(* Logix 5000 project; controller cal1632 1756-L62 rev 16.20; software revision 16.05; part 38 of 61 *)
(* tags used below, declared in another part *)
   p23r17 : routine;
   FAULT : BOOL;
   HMI : BOOL;
   p01r09_pb_global_reset : BOOL;
   p02_real_from_hmi : hmi_real;
   p23_ai_lfl : REAL;
   p23_ai_metering_roll_amps : REAL;
   p23_ai_metering_roll_hz : REAL;
   p23_ai_metering_roll_speed_fpm : REAL;
   p23_ai_prs : REAL;
   p23_ai_servo_ds_position : REAL;
   p23_ai_servo_ds_torque : REAL;
   p23_ai_servo_os_position : REAL;
   p23_ai_servo_os_torque : REAL;
   p23_ai_servo_os_velocity : REAL;
   p23_ai_supply_amps : REAL;
   p23_ai_supply_hz : REAL;
   p23_ai_supply_rpm : REAL;
   p23_dint_to_hmi : DINT[32];
   p23_param_lfl_hhl : REAL;
   p23_param_lfl_hl : REAL;
   p23_param_zone_pressure : REAL;
   p23_real_to_hmi : REAL[112];
   p23r02 : routine;
   p23r06 : routine;
   p23r06_timer_fault : TIMER[4];
   p23r06_timer_warning : TIMER[4];
   p23r07 : routine;
   p23r07_timer_fault : TIMER[4];
   p23r07_timer_warning : TIMER[4];
   p23r08 : routine;
   p23r08_timer_fault : TIMER[4];
   p23r08_timer_warning : TIMER[4];
   p23r11 : routine;
   p23r12 : routine;
   p23r13 : routine;
   p23r15 : routine;
(* P23_Impreg, continued *)

ROUTINE R06_Real_to_HMI   (* ladder *)
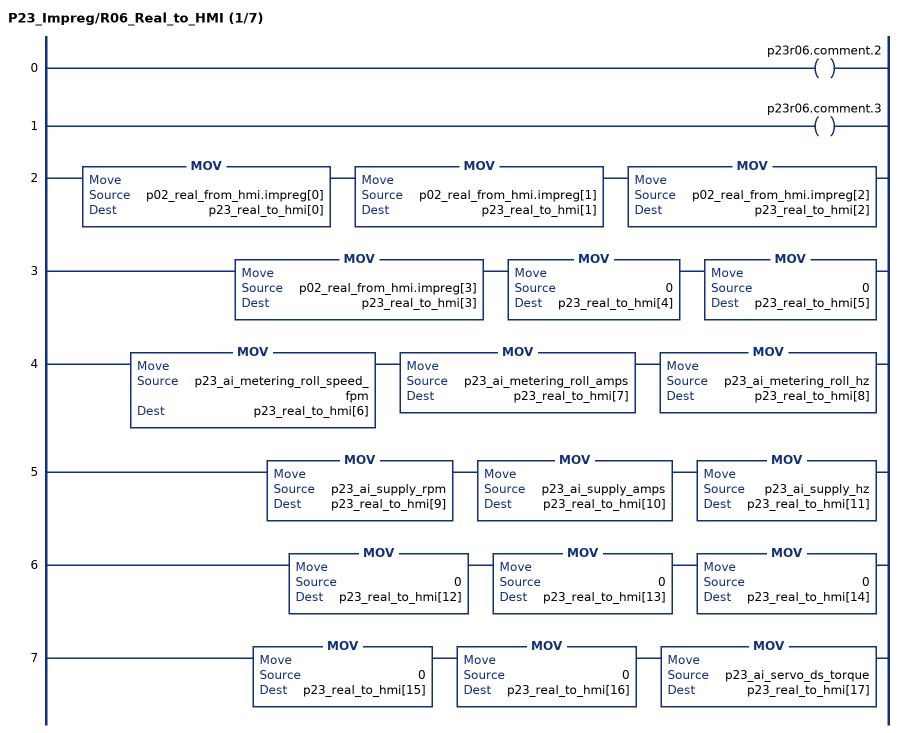
   0: OTE(p23r06.comment.2);
   1: OTE(p23r06.comment.3);
   2: MOV(p02_real_from_hmi.impreg[0],p23_real_to_hmi[0])MOV(p02_real_from_hmi.impreg[1],p23_real_to_hmi[1])MOV(p02_real_from_hmi.impreg[2],p23_real_to_hmi[2]);
   3: MOV(p02_real_from_hmi.impreg[3],p23_real_to_hmi[3])MOV(0,p23_real_to_hmi[4])MOV(0,p23_real_to_hmi[5]);
   4: MOV(p23_ai_metering_roll_speed_fpm,p23_real_to_hmi[6])MOV(p23_ai_metering_roll_amps,p23_real_to_hmi[7])MOV(p23_ai_metering_roll_hz,p23_real_to_hmi[8]);
   5: MOV(p23_ai_supply_rpm,p23_real_to_hmi[9])MOV(p23_ai_supply_amps,p23_real_to_hmi[10])MOV(p23_ai_supply_hz,p23_real_to_hmi[11]);
   6: MOV(0,p23_real_to_hmi[12])MOV(0,p23_real_to_hmi[13])MOV(0,p23_real_to_hmi[14]);
   7: MOV(0,p23_real_to_hmi[15])MOV(0,p23_real_to_hmi[16])MOV(p23_ai_servo_ds_torque,p23_real_to_hmi[17]);
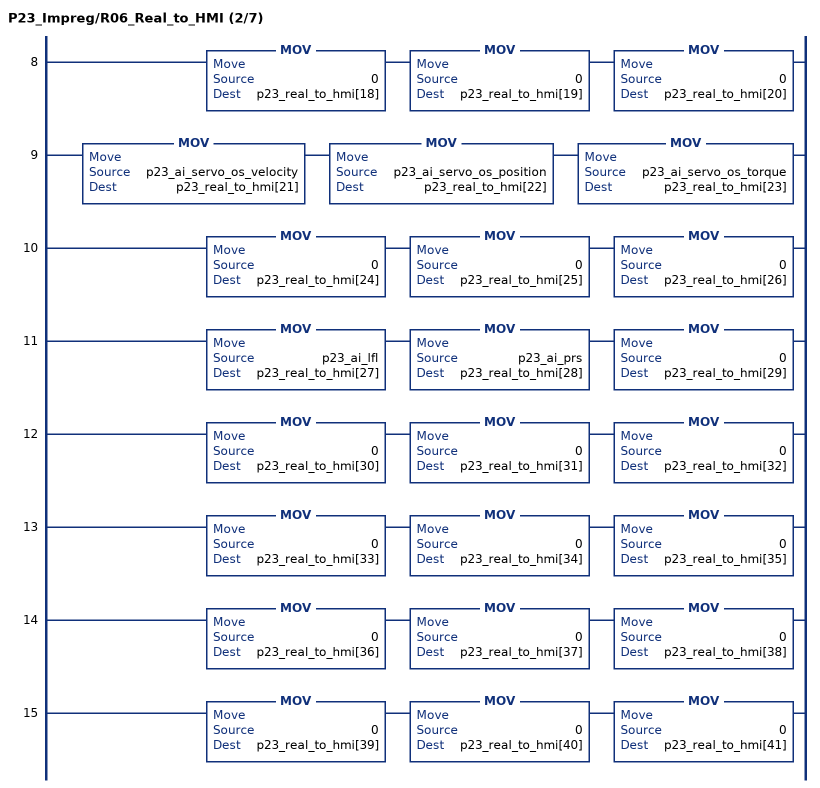
   8: MOV(0,p23_real_to_hmi[18])MOV(0,p23_real_to_hmi[19])MOV(0,p23_real_to_hmi[20]);
   9: MOV(p23_ai_servo_os_velocity,p23_real_to_hmi[21])MOV(p23_ai_servo_os_position,p23_real_to_hmi[22])MOV(p23_ai_servo_os_torque,p23_real_to_hmi[23]);
   10: MOV(0,p23_real_to_hmi[24])MOV(0,p23_real_to_hmi[25])MOV(0,p23_real_to_hmi[26]);
   11: MOV(p23_ai_lfl,p23_real_to_hmi[27])MOV(p23_ai_prs,p23_real_to_hmi[28])MOV(0,p23_real_to_hmi[29]);
   12: MOV(0,p23_real_to_hmi[30])MOV(0,p23_real_to_hmi[31])MOV(0,p23_real_to_hmi[32]);
   13: MOV(0,p23_real_to_hmi[33])MOV(0,p23_real_to_hmi[34])MOV(0,p23_real_to_hmi[35]);
   14: MOV(0,p23_real_to_hmi[36])MOV(0,p23_real_to_hmi[37])MOV(0,p23_real_to_hmi[38]);
   15: MOV(0,p23_real_to_hmi[39])MOV(0,p23_real_to_hmi[40])MOV(0,p23_real_to_hmi[41]);
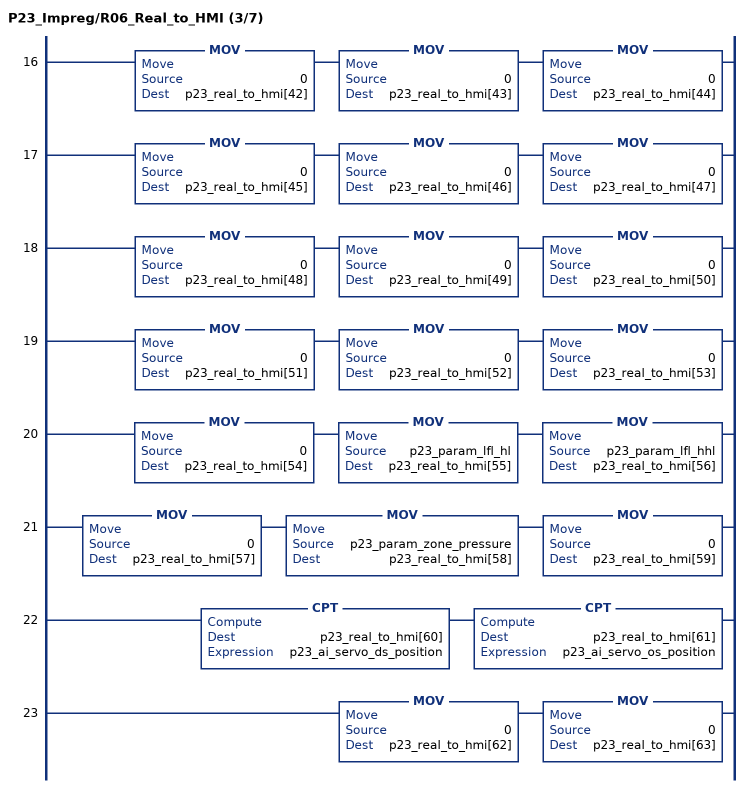
   16: MOV(0,p23_real_to_hmi[42])MOV(0,p23_real_to_hmi[43])MOV(0,p23_real_to_hmi[44]);
   17: MOV(0,p23_real_to_hmi[45])MOV(0,p23_real_to_hmi[46])MOV(0,p23_real_to_hmi[47]);
   18: MOV(0,p23_real_to_hmi[48])MOV(0,p23_real_to_hmi[49])MOV(0,p23_real_to_hmi[50]);
   19: MOV(0,p23_real_to_hmi[51])MOV(0,p23_real_to_hmi[52])MOV(0,p23_real_to_hmi[53]);
   20: MOV(0,p23_real_to_hmi[54])MOV(p23_param_lfl_hl,p23_real_to_hmi[55])MOV(p23_param_lfl_hhl,p23_real_to_hmi[56]);
   21: MOV(0,p23_real_to_hmi[57])MOV(p23_param_zone_pressure,p23_real_to_hmi[58])MOV(0,p23_real_to_hmi[59]);
   22: CPT(p23_real_to_hmi[60],p23_ai_servo_ds_position)CPT(p23_real_to_hmi[61],p23_ai_servo_os_position);
   23: MOV(0,p23_real_to_hmi[62])MOV(0,p23_real_to_hmi[63]);
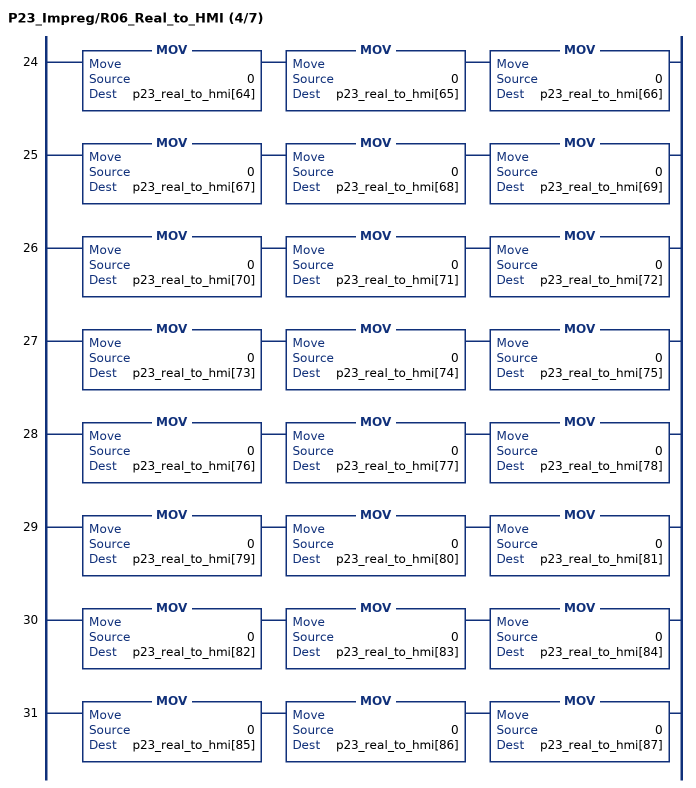
   24: MOV(0,p23_real_to_hmi[64])MOV(0,p23_real_to_hmi[65])MOV(0,p23_real_to_hmi[66]);
   25: MOV(0,p23_real_to_hmi[67])MOV(0,p23_real_to_hmi[68])MOV(0,p23_real_to_hmi[69]);
   26: MOV(0,p23_real_to_hmi[70])MOV(0,p23_real_to_hmi[71])MOV(0,p23_real_to_hmi[72]);
   27: MOV(0,p23_real_to_hmi[73])MOV(0,p23_real_to_hmi[74])MOV(0,p23_real_to_hmi[75]);
   28: MOV(0,p23_real_to_hmi[76])MOV(0,p23_real_to_hmi[77])MOV(0,p23_real_to_hmi[78]);
   29: MOV(0,p23_real_to_hmi[79])MOV(0,p23_real_to_hmi[80])MOV(0,p23_real_to_hmi[81]);
   30: MOV(0,p23_real_to_hmi[82])MOV(0,p23_real_to_hmi[83])MOV(0,p23_real_to_hmi[84]);
   31: MOV(0,p23_real_to_hmi[85])MOV(0,p23_real_to_hmi[86])MOV(0,p23_real_to_hmi[87]);
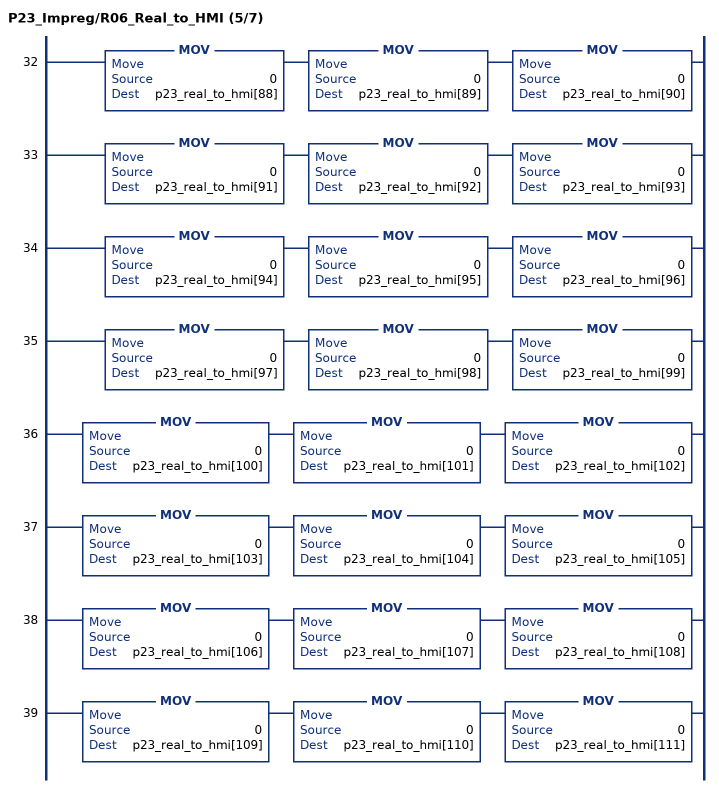
   32: MOV(0,p23_real_to_hmi[88])MOV(0,p23_real_to_hmi[89])MOV(0,p23_real_to_hmi[90]);
   33: MOV(0,p23_real_to_hmi[91])MOV(0,p23_real_to_hmi[92])MOV(0,p23_real_to_hmi[93]);
   34: MOV(0,p23_real_to_hmi[94])MOV(0,p23_real_to_hmi[95])MOV(0,p23_real_to_hmi[96]);
   35: MOV(0,p23_real_to_hmi[97])MOV(0,p23_real_to_hmi[98])MOV(0,p23_real_to_hmi[99]);
   36: MOV(0,p23_real_to_hmi[100])MOV(0,p23_real_to_hmi[101])MOV(0,p23_real_to_hmi[102]);
   37: MOV(0,p23_real_to_hmi[103])MOV(0,p23_real_to_hmi[104])MOV(0,p23_real_to_hmi[105]);
   38: MOV(0,p23_real_to_hmi[106])MOV(0,p23_real_to_hmi[107])MOV(0,p23_real_to_hmi[108]);
   39: MOV(0,p23_real_to_hmi[109])MOV(0,p23_real_to_hmi[110])MOV(0,p23_real_to_hmi[111]);
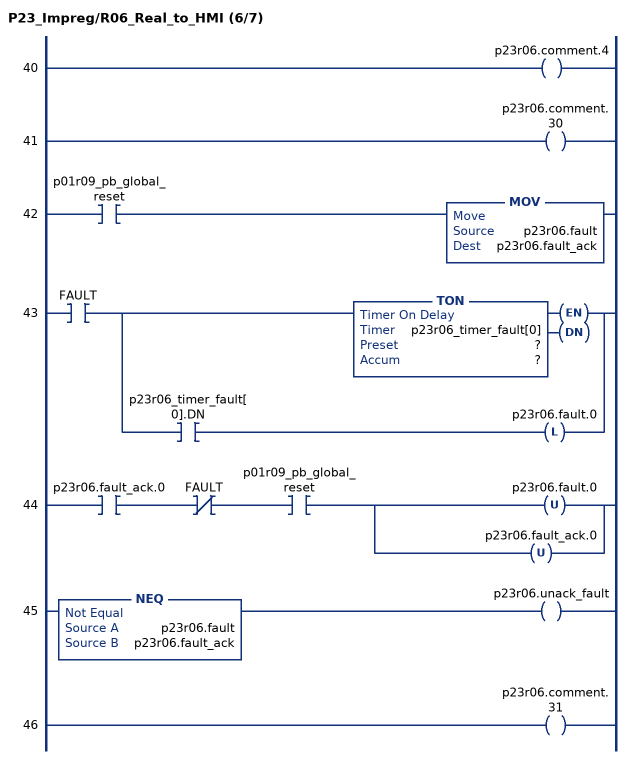
   40: OTE(p23r06.comment.4);
   41: OTE(p23r06.comment.30);
   42: XIC(p01r09_pb_global_reset)MOV(p23r06.fault,p23r06.fault_ack);
   43: XIC(FAULT)[TON(p23r06_timer_fault[0],?,?) ,XIC(p23r06_timer_fault[0].DN) OTL(p23r06.fault.0) ];
   44: XIC(p23r06.fault_ack.0)XIO(FAULT)XIC(p01r09_pb_global_reset)[OTU(p23r06.fault.0) ,OTU(p23r06.fault_ack.0) ];
   45: NEQ(p23r06.fault,p23r06.fault_ack)OTE(p23r06.unack_fault);
   46: OTE(p23r06.comment.31);
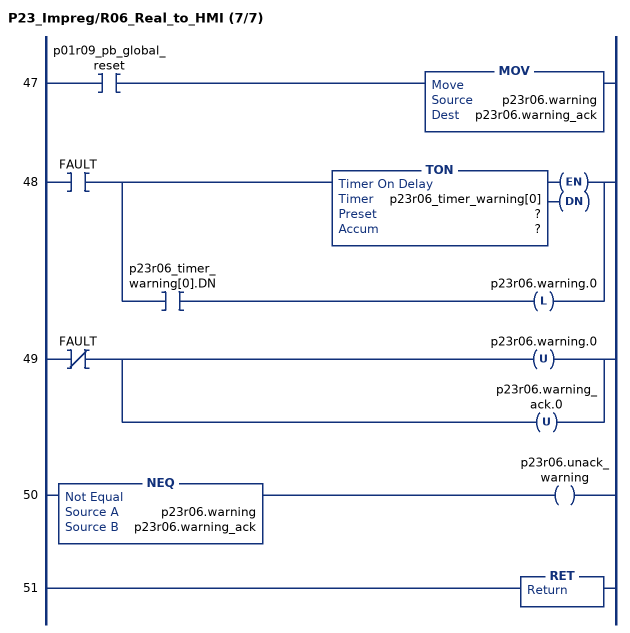
   47: XIC(p01r09_pb_global_reset)MOV(p23r06.warning,p23r06.warning_ack);
   48: XIC(FAULT)[TON(p23r06_timer_warning[0],?,?) ,XIC(p23r06_timer_warning[0].DN) OTL(p23r06.warning.0) ];
   49: XIO(FAULT)[OTU(p23r06.warning.0) ,OTU(p23r06.warning_ack.0) ];
   50: NEQ(p23r06.warning,p23r06.warning_ack)OTE(p23r06.unack_warning);
   51: RET();
END_ROUTINE

ROUTINE R07_Alarms   (* ladder *)
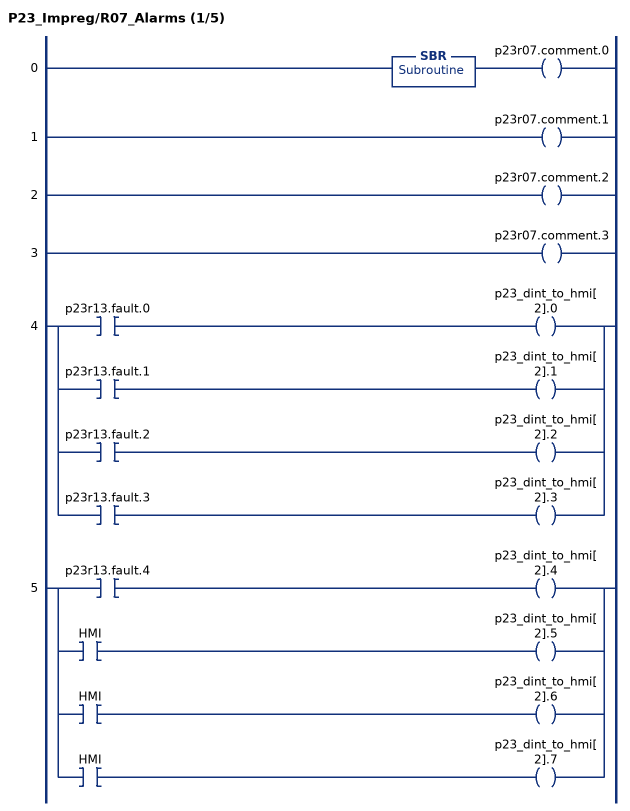
   0: SBR()OTE(p23r07.comment.0);
   1: OTE(p23r07.comment.1);
   2: OTE(p23r07.comment.2);
   3: OTE(p23r07.comment.3);
   4: [XIC(p23r13.fault.0) OTE(p23_dint_to_hmi[2].0) ,XIC(p23r13.fault.1) OTE(p23_dint_to_hmi[2].1) ,XIC(p23r13.fault.2) OTE(p23_dint_to_hmi[2].2) ,XIC(p23r13.fault.3) OTE(p23_dint_to_hmi[2].3) ];
   5: [XIC(p23r13.fault.4) OTE(p23_dint_to_hmi[2].4) ,XIC(HMI) OTE(p23_dint_to_hmi[2].5) ,XIC(HMI) OTE(p23_dint_to_hmi[2].6) ,XIC(HMI) OTE(p23_dint_to_hmi[2].7) ];
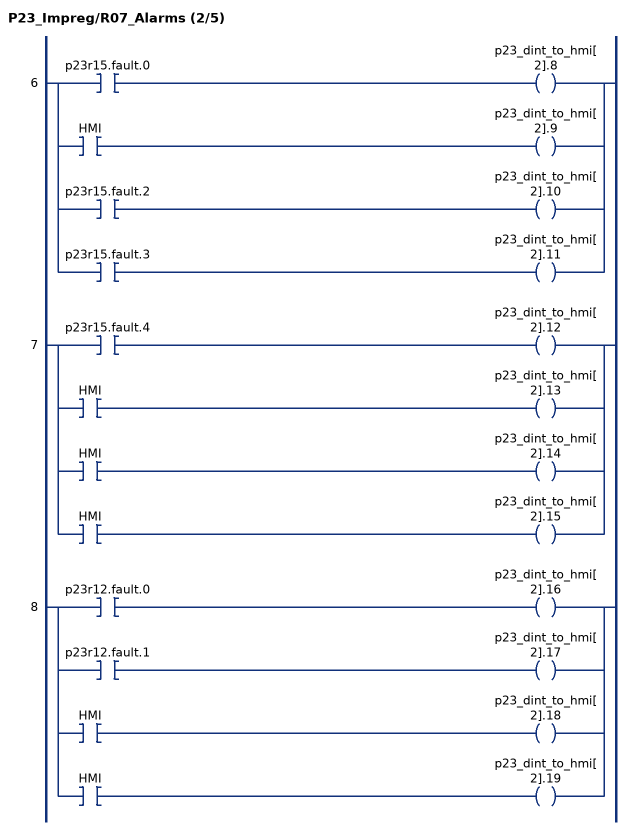
   6: [XIC(p23r15.fault.0) OTE(p23_dint_to_hmi[2].8) ,XIC(HMI) OTE(p23_dint_to_hmi[2].9) ,XIC(p23r15.fault.2) OTE(p23_dint_to_hmi[2].10) ,XIC(p23r15.fault.3) OTE(p23_dint_to_hmi[2].11) ];
   7: [XIC(p23r15.fault.4) OTE(p23_dint_to_hmi[2].12) ,XIC(HMI) OTE(p23_dint_to_hmi[2].13) ,XIC(HMI) OTE(p23_dint_to_hmi[2].14) ,XIC(HMI) OTE(p23_dint_to_hmi[2].15) ];
   8: [XIC(p23r12.fault.0) OTE(p23_dint_to_hmi[2].16) ,XIC(p23r12.fault.1) OTE(p23_dint_to_hmi[2].17) ,XIC(HMI) OTE(p23_dint_to_hmi[2].18) ,XIC(HMI) OTE(p23_dint_to_hmi[2].19) ];
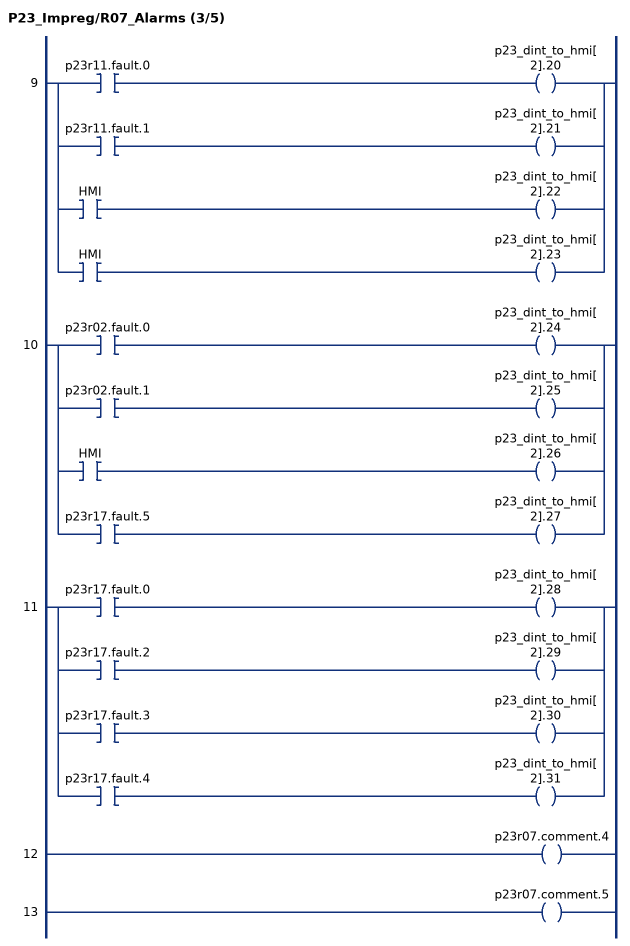
   9: [XIC(p23r11.fault.0) OTE(p23_dint_to_hmi[2].20) ,XIC(p23r11.fault.1) OTE(p23_dint_to_hmi[2].21) ,XIC(HMI) OTE(p23_dint_to_hmi[2].22) ,XIC(HMI) OTE(p23_dint_to_hmi[2].23) ];
   10: [XIC(p23r02.fault.0) OTE(p23_dint_to_hmi[2].24) ,XIC(p23r02.fault.1) OTE(p23_dint_to_hmi[2].25) ,XIC(HMI) OTE(p23_dint_to_hmi[2].26) ,XIC(p23r17.fault.5) OTE(p23_dint_to_hmi[2].27) ];
   11: [XIC(p23r17.fault.0) OTE(p23_dint_to_hmi[2].28) ,XIC(p23r17.fault.2) OTE(p23_dint_to_hmi[2].29) ,XIC(p23r17.fault.3) OTE(p23_dint_to_hmi[2].30) ,XIC(p23r17.fault.4) OTE(p23_dint_to_hmi[2].31) ];
   12: OTE(p23r07.comment.4);
   13: OTE(p23r07.comment.5);
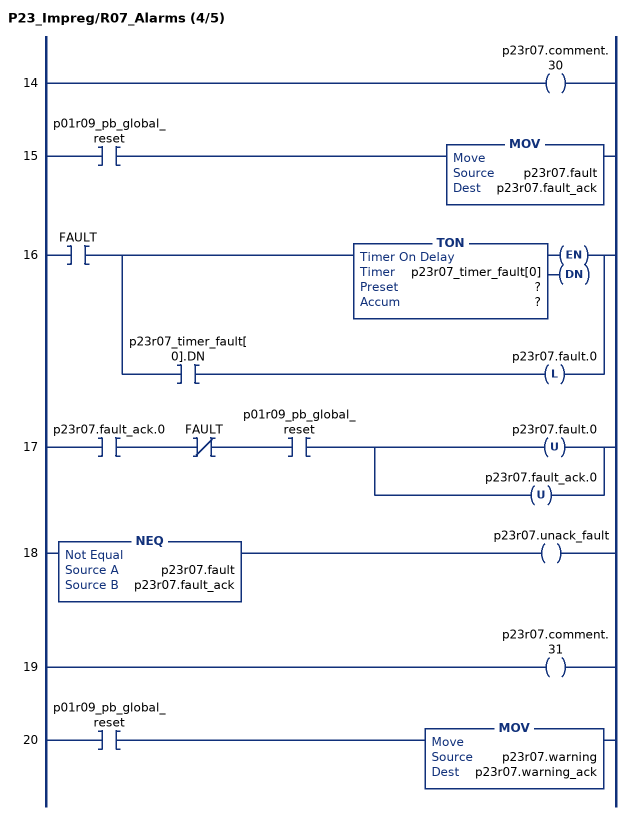
   14: OTE(p23r07.comment.30);
   15: XIC(p01r09_pb_global_reset)MOV(p23r07.fault,p23r07.fault_ack);
   16: XIC(FAULT)[TON(p23r07_timer_fault[0],?,?) ,XIC(p23r07_timer_fault[0].DN) OTL(p23r07.fault.0) ];
   17: XIC(p23r07.fault_ack.0)XIO(FAULT)XIC(p01r09_pb_global_reset)[OTU(p23r07.fault.0) ,OTU(p23r07.fault_ack.0) ];
   18: NEQ(p23r07.fault,p23r07.fault_ack)OTE(p23r07.unack_fault);
   19: OTE(p23r07.comment.31);
   20: XIC(p01r09_pb_global_reset)MOV(p23r07.warning,p23r07.warning_ack);
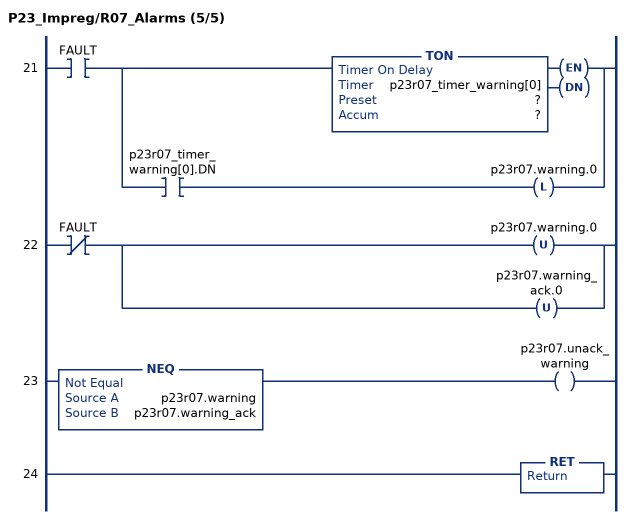
   21: XIC(FAULT)[TON(p23r07_timer_warning[0],?,?) ,XIC(p23r07_timer_warning[0].DN) OTL(p23r07.warning.0) ];
   22: XIO(FAULT)[OTU(p23r07.warning.0) ,OTU(p23r07.warning_ack.0) ];
   23: NEQ(p23r07.warning,p23r07.warning_ack)OTE(p23r07.unack_warning);
   24: RET();
END_ROUTINE

ROUTINE R08_Warnings   (* ladder *)
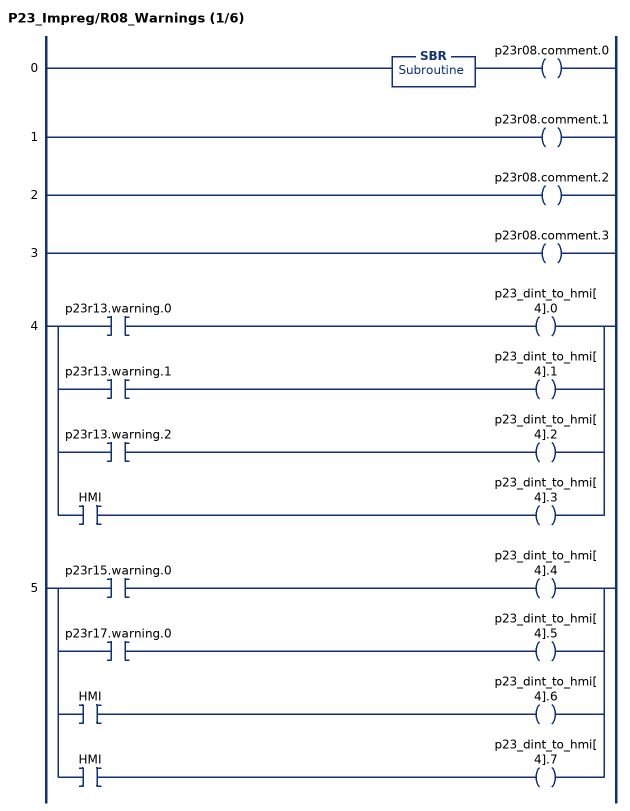
   0: SBR()OTE(p23r08.comment.0);
   1: OTE(p23r08.comment.1);
   2: OTE(p23r08.comment.2);
   3: OTE(p23r08.comment.3);
   4: [XIC(p23r13.warning.0) OTE(p23_dint_to_hmi[4].0) ,XIC(p23r13.warning.1) OTE(p23_dint_to_hmi[4].1) ,XIC(p23r13.warning.2) OTE(p23_dint_to_hmi[4].2) ,XIC(HMI) OTE(p23_dint_to_hmi[4].3) ];
   5: [XIC(p23r15.warning.0) OTE(p23_dint_to_hmi[4].4) ,XIC(p23r17.warning.0) OTE(p23_dint_to_hmi[4].5) ,XIC(HMI) OTE(p23_dint_to_hmi[4].6) ,XIC(HMI) OTE(p23_dint_to_hmi[4].7) ];
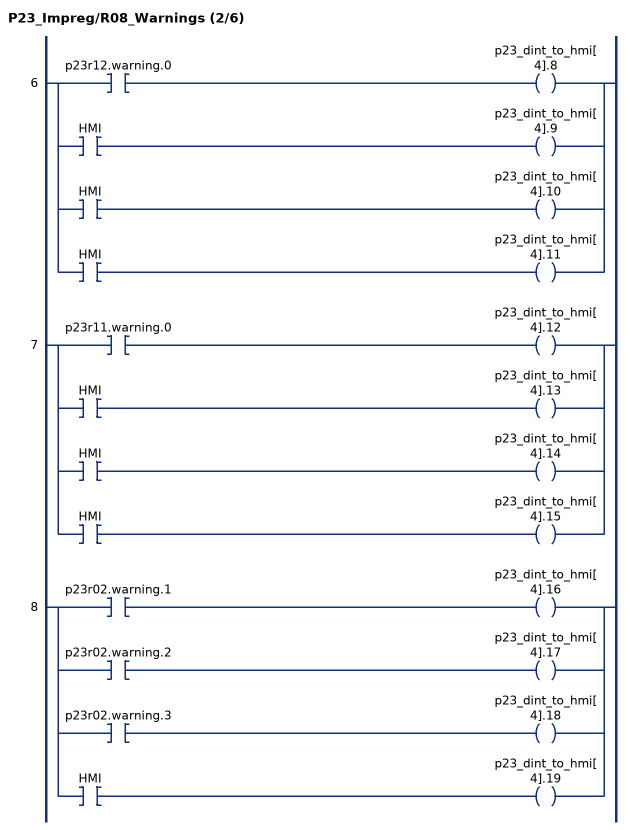
   6: [XIC(p23r12.warning.0) OTE(p23_dint_to_hmi[4].8) ,XIC(HMI) OTE(p23_dint_to_hmi[4].9) ,XIC(HMI) OTE(p23_dint_to_hmi[4].10) ,XIC(HMI) OTE(p23_dint_to_hmi[4].11) ];
   7: [XIC(p23r11.warning.0) OTE(p23_dint_to_hmi[4].12) ,XIC(HMI) OTE(p23_dint_to_hmi[4].13) ,XIC(HMI) OTE(p23_dint_to_hmi[4].14) ,XIC(HMI) OTE(p23_dint_to_hmi[4].15) ];
   8: [XIC(p23r02.warning.1) OTE(p23_dint_to_hmi[4].16) ,XIC(p23r02.warning.2) OTE(p23_dint_to_hmi[4].17) ,XIC(p23r02.warning.3) OTE(p23_dint_to_hmi[4].18) ,XIC(HMI) OTE(p23_dint_to_hmi[4].19) ];
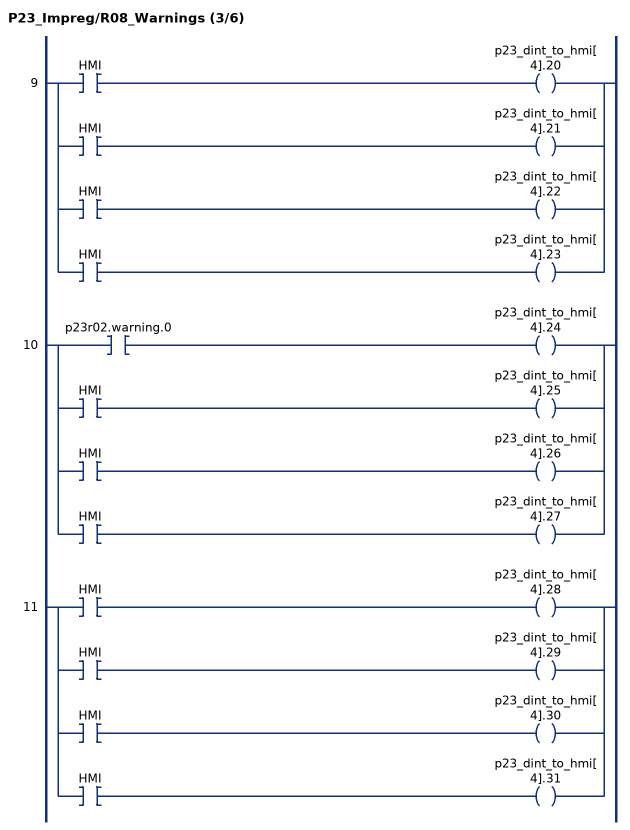
   9: [XIC(HMI) OTE(p23_dint_to_hmi[4].20) ,XIC(HMI) OTE(p23_dint_to_hmi[4].21) ,XIC(HMI) OTE(p23_dint_to_hmi[4].22) ,XIC(HMI) OTE(p23_dint_to_hmi[4].23) ];
   10: [XIC(p23r02.warning.0) OTE(p23_dint_to_hmi[4].24) ,XIC(HMI) OTE(p23_dint_to_hmi[4].25) ,XIC(HMI) OTE(p23_dint_to_hmi[4].26) ,XIC(HMI) OTE(p23_dint_to_hmi[4].27) ];
   11: [XIC(HMI) OTE(p23_dint_to_hmi[4].28) ,XIC(HMI) OTE(p23_dint_to_hmi[4].29) ,XIC(HMI) OTE(p23_dint_to_hmi[4].30) ,XIC(HMI) OTE(p23_dint_to_hmi[4].31) ];
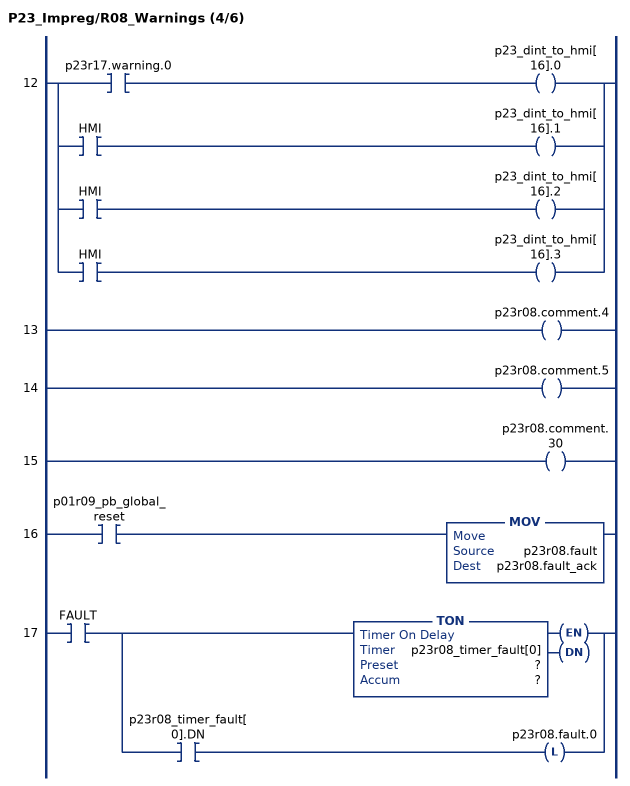
   12: [XIC(p23r17.warning.0) OTE(p23_dint_to_hmi[16].0) ,XIC(HMI) OTE(p23_dint_to_hmi[16].1) ,XIC(HMI) OTE(p23_dint_to_hmi[16].2) ,XIC(HMI) OTE(p23_dint_to_hmi[16].3) ];
   13: OTE(p23r08.comment.4);
   14: OTE(p23r08.comment.5);
   15: OTE(p23r08.comment.30);
   16: XIC(p01r09_pb_global_reset)MOV(p23r08.fault,p23r08.fault_ack);
   17: XIC(FAULT)[TON(p23r08_timer_fault[0],?,?) ,XIC(p23r08_timer_fault[0].DN) OTL(p23r08.fault.0) ];
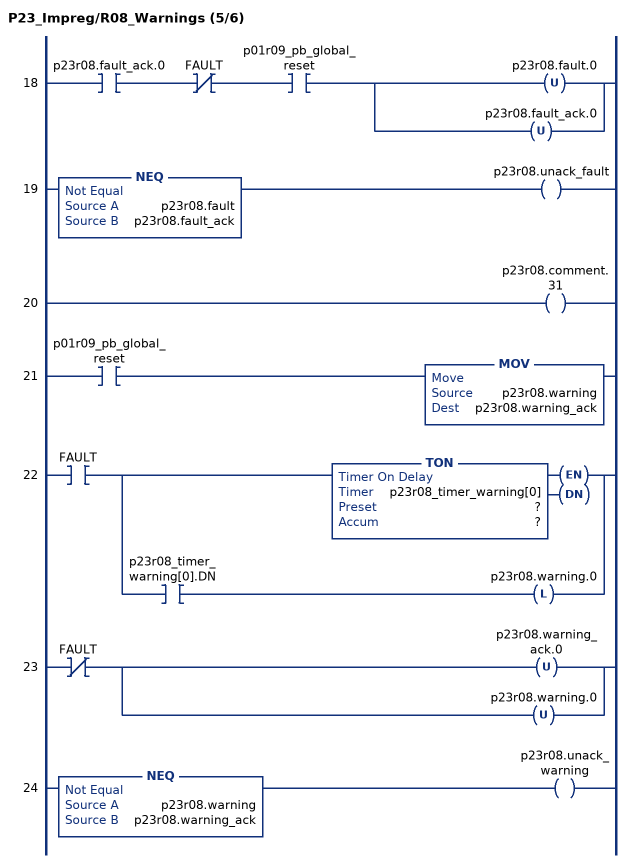
   18: XIC(p23r08.fault_ack.0)XIO(FAULT)XIC(p01r09_pb_global_reset)[OTU(p23r08.fault.0) ,OTU(p23r08.fault_ack.0) ];
   19: NEQ(p23r08.fault,p23r08.fault_ack)OTE(p23r08.unack_fault);
   20: OTE(p23r08.comment.31);
   21: XIC(p01r09_pb_global_reset)MOV(p23r08.warning,p23r08.warning_ack);
   22: XIC(FAULT)[TON(p23r08_timer_warning[0],?,?) ,XIC(p23r08_timer_warning[0].DN) OTL(p23r08.warning.0) ];
   23: XIO(FAULT)[OTU(p23r08.warning_ack.0) ,OTU(p23r08.warning.0) ];
   24: NEQ(p23r08.warning,p23r08.warning_ack)OTE(p23r08.unack_warning);
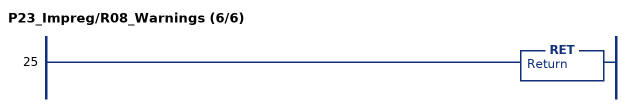
   25: RET();
END_ROUTINE
